(* IEC 61131-3 sources: CodesysTest/export/SX_1195.dev/Plc Logic/Application/PRJ Specific/1195 Testing/Clamping Mechanism/FB_ClampingMechanism.pou/Ready.prop, 1 file *)

(* ---- Get.pm.st ---- *)
(*#-#-#-#-#-#-#-#-#-#---Declaration---#-#-#-#-#-#-#-#-#-#-#-#-#*)

VAR
END_VAR
(*#-#-#-#-#-#-#-#-#-#---Implementation---#-#-#-#-#-#-#-#-#-#-#-#-#*)

Ready:=_ready;
